Yaskawa INFORM job: u_incl_braTRJ0.JBI

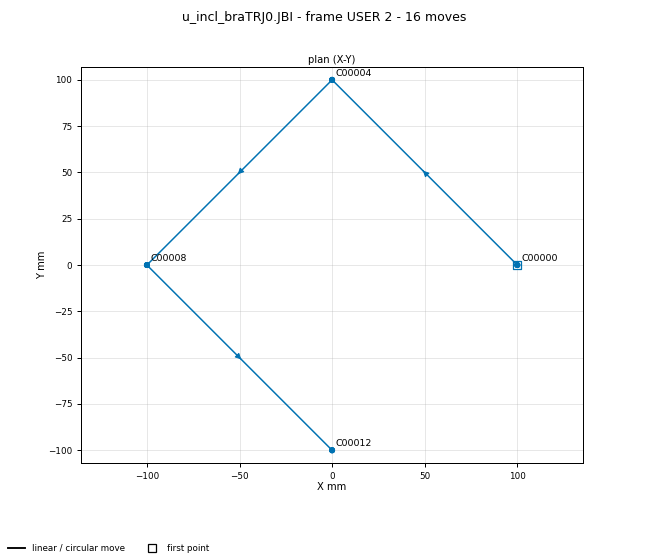
[picture p0: tool path of u_incl_braTRJ0.JBI in frame USER 2, 16 of 16 moves have a stored position in this frame; points joined in program order, loops and branches not executed]
/JOB
//NAME u_incl_braTRJ0
///FOLDERNAME DEMO
//POS
///NPOS 16,0,0,0,0,0
///USER 2
///TOOL 7
///POSTYPE USER
///RECTAN
///RCONF 1,0,0,0,0,0,0,0,0,0,0,0,0,0,0,0,0,0,0,0,0,0,0,0
C00000=100.000,0.000,20.000,-180.0000,-20.0125,0.0000
C00001=100.000,0.000,20.000,-159.9875,0.0000,0.0000
C00002=100.000,0.000,20.000,-180.0000,20.0125,0.0000
C00003=100.000,0.000,20.000,159.9875,0.0000,0.0000
C00004=0.000,100.000,20.000,-180.0000,-20.0125,0.0000
C00005=0.000,100.000,20.000,-159.9875,0.0000,0.0000
C00006=0.000,100.000,20.000,-180.0000,20.0125,0.0000
C00007=0.000,100.000,20.000,159.9875,0.0000,0.0000
C00008=-100.000,0.000,20.000,-180.0000,-20.0125,0.0000
C00009=-100.000,0.000,20.000,-159.9875,0.0000,0.0000
C00010=-100.000,0.000,20.000,-180.0000,20.0125,0.0000
C00011=-100.000,0.000,20.000,159.9875,0.0000,0.0000
C00012=0.000,-100.000,20.000,-180.0000,-20.0125,0.0000
C00013=0.000,-100.000,20.000,-159.9875,0.0000,0.0000
C00014=0.000,-100.000,20.000,-180.0000,20.0125,0.0000
C00015=0.000,-100.000,20.000,159.9875,0.0000,0.0000
//INST
///DATE 2022/04/08 11:28
///COMM
///ATTR SC,RW,RJ
////FRAME USER 2
///GROUP1 RB1
NOP
SPEED V=10.0
MOVL C00000
MOVL C00001
MOVL C00002
MOVL C00003
MOVL C00004
MOVL C00005
MOVL C00006
MOVL C00007
MOVL C00008
MOVL C00009
MOVL C00010
MOVL C00011
MOVL C00012
MOVL C00013
MOVL C00014
MOVL C00015
END
